Fanuc KAREL source: NC0067.KL

-- PROVISIONAL review KL for V940-1; original PC SHA256 ae2f626e60705a0e145d5f72e343ff53052edb001488e1f967d241d2420f5ffe
-- Incomplete behavior may be omitted. Consult companion uncertainty JSON. Do not deploy.
PROGRAM NC0067
%NOLOCKGROUP
-- UNRESOLVED_LOCAL_POOL 11 cells at code offset 3; source declarations unknown
-- DIRECT_LOCAL_WORD_ACCESS alone does not prove INTEGER, REAL, or BOOLEAN
BEGIN
  -- V9_EXPOSED_INDEXED_TABLE_HINT layout=0001; 20 counted words exposed once; source arms/runtime held
  -- V9_FOOTER_20_HINT 10 numerical footer links; VM transfer unproved
  -- UNRESOLVED_PC offsets 0-8; opcodes 2B,2C,7B
  -- UNRESOLVED_PC offsets 13-20; opcodes 9D,23
  -- UNRESOLVED_PC offsets 25-54; opcodes 9D,23,9E,2E,22,7A
  -- UNRESOLVED_PC offsets 59-88; opcodes 9D,23,9E,2E,22,7A
  -- UNRESOLVED_PC offsets 93-122; opcodes 9D,23,9E,2E,22,7A
  -- UNRESOLVED_PC offsets 127-156; opcodes 9D,23,9E,2E,22,7A
  -- UNRESOLVED_PC offsets 161-190; opcodes 9D,23,9E,2E,22,7A
  -- UNRESOLVED_PC offsets 195-224; opcodes 9D,23,9E,2E,22,7A
  -- UNRESOLVED_PC offsets 229-258; opcodes 9D,23,9E,2E,22,7A
  -- UNRESOLVED_PC offsets 263-292; opcodes 9D,23,9E,2E,22,7A
  -- UNRESOLVED_PC offsets 297-326; opcodes 9D,23,9E,2E,22,7A
  -- UNRESOLVED_PC offsets 331-360; opcodes 9D,23,9E,2E,22,7A
  -- UNRESOLVED_PC offsets 365-379; opcodes 21,9D,52,23
  -- UNRESOLVED_PC offsets 384-399; opcodes 20,2C,23
  -- UNRESOLVED_PC offsets 404-419; opcodes 20,2C,23
  -- UNRESOLVED_PC offsets 424-439; opcodes 20,2C,23
  -- UNRESOLVED_PC offsets 444-459; opcodes 20,2C,23
  -- UNRESOLVED_PC offsets 464-479; opcodes 20,2C,23
  -- UNRESOLVED_PC offsets 484-499; opcodes 20,2C,23
  -- UNRESOLVED_PC offsets 504-519; opcodes 20,2C,23
  -- UNRESOLVED_PC offsets 524-539; opcodes 20,2C,23
  -- UNRESOLVED_PC offsets 544-559; opcodes 20,2C,23
  -- UNRESOLVED_PC offsets 564-579; opcodes 20,2C,23
  -- UNRESOLVED_PC offsets 584-588; opcodes 7F
  -- UNRESOLVED_PC offsets 593-597; opcodes 27,AA
  -- UNRESOLVED_PC offsets 602-606; opcodes 7F
END NC0067
